PROGRAM MAIN
VAR
END_VAR

END_PROGRAM

(* stored: Version 1.1.0.1
   POU MAIN: Id {726c3a48-09c4-43f6-8118-c078e9ae3b3a} *)
